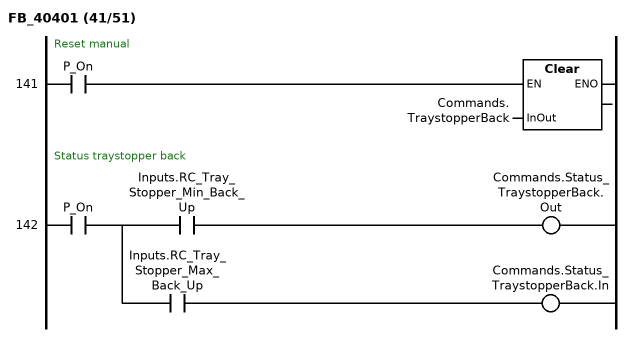
(* [picture p174: FB_40401, rungs 141-142] *)
(* Rung 141: Reset manual *)
IF P_On THEN Clear(InOut := Commands.TraystopperBack); END_IF;
(* Rung 142: Status traystopper back *)
Commands.Status_TraystopperBack.Out := P_On AND Inputs.RC_Tray_Stopper_Min_Back_Up;
Commands.Status_TraystopperBack.In := P_On AND Inputs.RC_Tray_Stopper_Max_Back_Up;

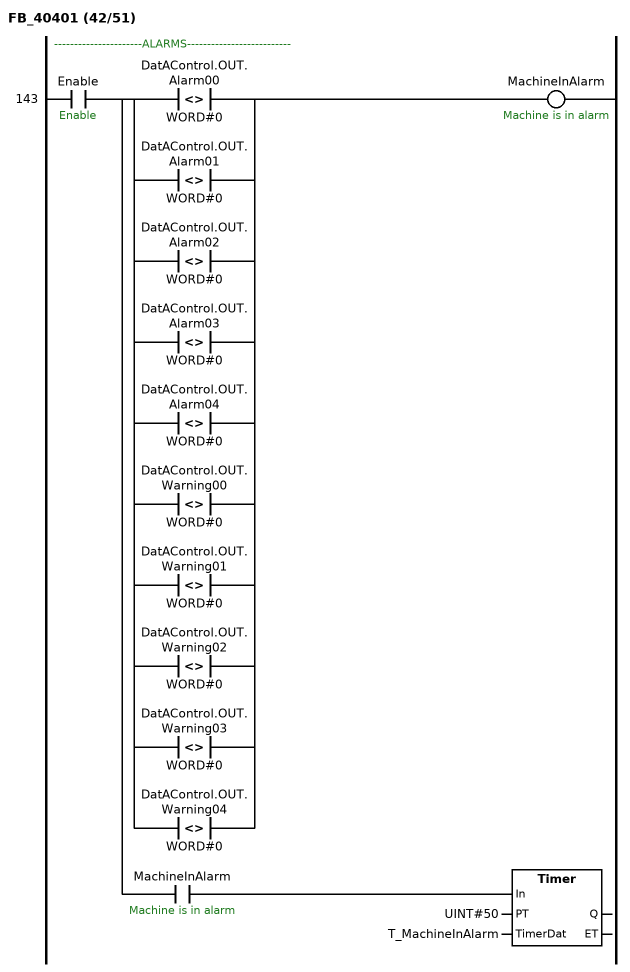
(* Rung 143: ----------------------ALARMS-------------------------- *)
MachineInAlarm := Enable AND ((DatAControl.OUT.Alarm00 <> WORD#0) OR (DatAControl.OUT.Alarm01 <> WORD#0) OR (DatAControl.OUT.Alarm02 <> WORD#0) OR (DatAControl.OUT.Alarm03 <> WORD#0) OR (DatAControl.OUT.Alarm04 <> WORD#0) OR (DatAControl.OUT.Warning00 <> WORD#0) OR (DatAControl.OUT.Warning01 <> WORD#0) OR (DatAControl.OUT.Warning02 <> WORD#0) OR (DatAControl.OUT.Warning03 <> WORD#0) OR (DatAControl.OUT.Warning04 <> WORD#0));
_t68 := Timer(In := Enable AND MachineInAlarm, PT := UINT#50, TimerDat := T_MachineInAlarm);

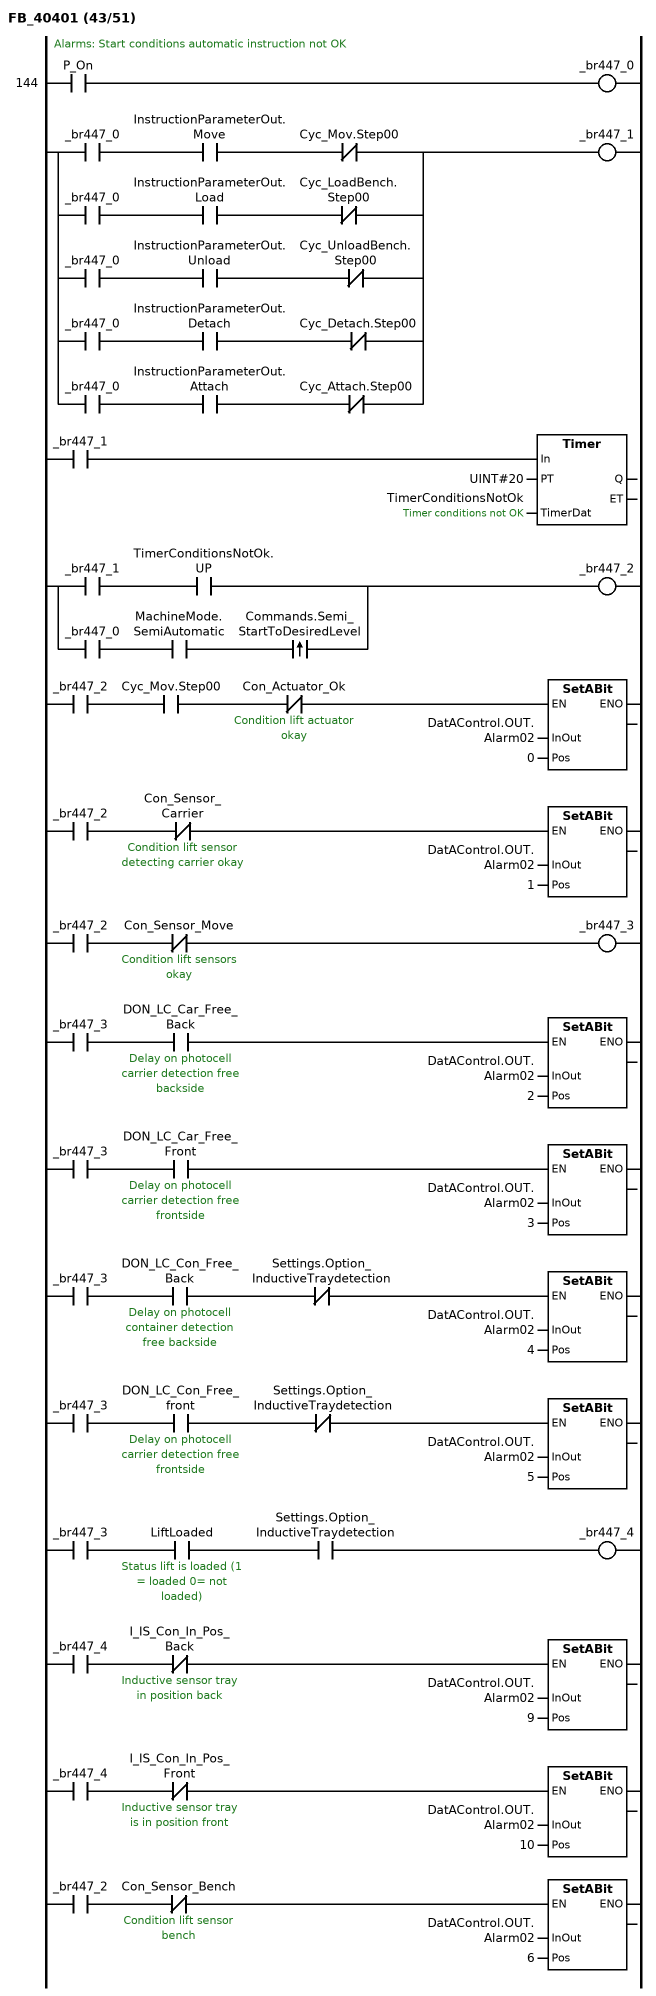
(* Rung 144: Alarms: Start conditions automatic instruction not OK *)
_br447_0 := P_On;
_br447_1 := (_br447_0 AND InstructionParameterOut.Move AND NOT Cyc_Mov.Step00) OR (_br447_0 AND InstructionParameterOut.Load AND NOT Cyc_LoadBench.Step00) OR (_br447_0 AND InstructionParameterOut.Unload AND NOT Cyc_UnloadBench.Step00) OR (_br447_0 AND InstructionParameterOut.Detach AND NOT Cyc_Detach.Step00) OR (_br447_0 AND InstructionParameterOut.Attach AND NOT Cyc_Attach.Step00);
_t69 := Timer(In := _br447_1, PT := UINT#20, TimerDat := TimerConditionsNotOk);
_e70(CLK := Commands.Semi_StartToDesiredLevel);
_br447_2 := (_br447_1 AND TimerConditionsNotOk.UP) OR (_br447_0 AND MachineMode.SemiAutomatic AND _e70.Q);
IF _br447_2 AND Cyc_Mov.Step00 AND NOT Con_Actuator_Ok THEN
    SetABit(InOut := DatAControl.OUT.Alarm02, Pos := 0);
END_IF;
IF _br447_2 AND NOT Con_Sensor_Carrier THEN SetABit(InOut := DatAControl.OUT.Alarm02, Pos := 1); END_IF;
_br447_3 := _br447_2 AND NOT Con_Sensor_Move;
IF _br447_3 AND DON_LC_Car_Free_Back THEN SetABit(InOut := DatAControl.OUT.Alarm02, Pos := 2); END_IF;
IF _br447_3 AND DON_LC_Car_Free_Front THEN SetABit(InOut := DatAControl.OUT.Alarm02, Pos := 3); END_IF;
IF _br447_3 AND DON_LC_Con_Free_Back AND NOT Settings.Option_InductiveTraydetection THEN
    SetABit(InOut := DatAControl.OUT.Alarm02, Pos := 4);
END_IF;
IF _br447_3 AND DON_LC_Con_Free_front AND NOT Settings.Option_InductiveTraydetection THEN
    SetABit(InOut := DatAControl.OUT.Alarm02, Pos := 5);
END_IF;
_br447_4 := _br447_3 AND LiftLoaded AND Settings.Option_InductiveTraydetection;
IF _br447_4 AND NOT I_IS_Con_In_Pos_Back THEN SetABit(InOut := DatAControl.OUT.Alarm02, Pos := 9); END_IF;
IF _br447_4 AND NOT I_IS_Con_In_Pos_Front THEN
    SetABit(InOut := DatAControl.OUT.Alarm02, Pos := 10);
END_IF;
IF _br447_2 AND NOT Con_Sensor_Bench THEN SetABit(InOut := DatAControl.OUT.Alarm02, Pos := 6); END_IF;

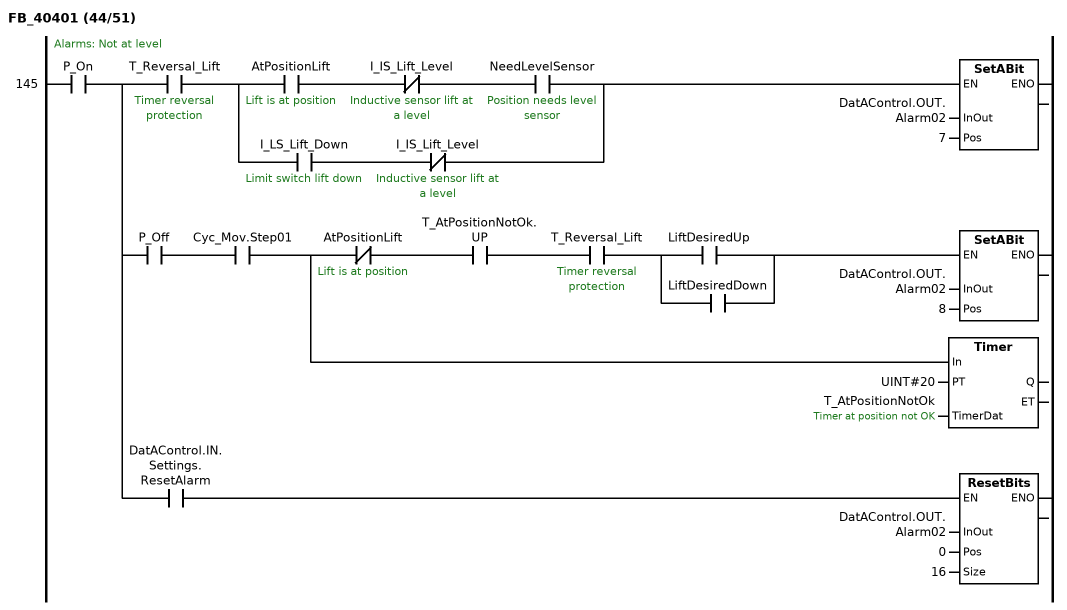
(* Rung 145: Alarms: Not at level *)
IF P_On AND T_Reversal_Lift AND ((AtPositionLift AND NOT I_IS_Lift_Level AND NeedLevelSensor) OR (I_LS_Lift_Down AND NOT I_IS_Lift_Level)) THEN
    SetABit(InOut := DatAControl.OUT.Alarm02, Pos := 7);
END_IF;
IF P_On AND P_Off AND Cyc_Mov.Step01 AND NOT AtPositionLift AND T_AtPositionNotOk.UP AND T_Reversal_Lift AND (LiftDesiredUp OR LiftDesiredDown) THEN
    SetABit(InOut := DatAControl.OUT.Alarm02, Pos := 8);
END_IF;
_t71 := Timer(In := P_On AND P_Off AND Cyc_Mov.Step01, PT := UINT#20, TimerDat := T_AtPositionNotOk);
IF P_On AND DatAControl.IN.Settings.ResetAlarm THEN
    ResetBits(InOut := DatAControl.OUT.Alarm02, Pos := 0, Size := 16);
END_IF;

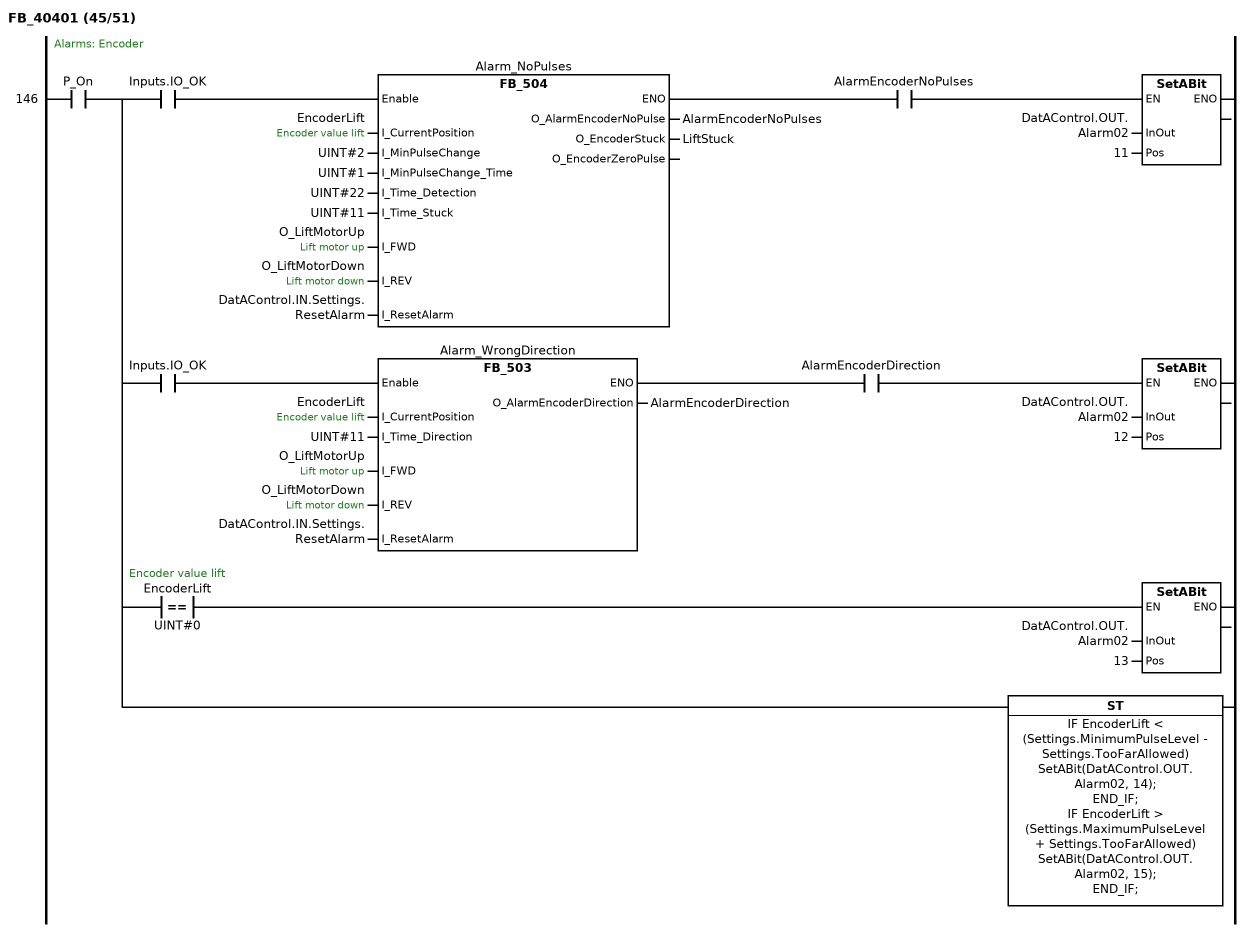
(* Rung 146: Alarms: Encoder *)
Alarm_NoPulses(Enable := P_On AND Inputs.IO_OK, I_CurrentPosition := EncoderLift, I_MinPulseChange := UINT#2, I_MinPulseChange_Time := UINT#1, I_Time_Detection := UINT#22, I_Time_Stuck := UINT#11, I_FWD := O_LiftMotorUp, I_REV := O_LiftMotorDown, I_ResetAlarm := DatAControl.IN.Settings.ResetAlarm, O_AlarmEncoderNoPulse => AlarmEncoderNoPulses, O_EncoderStuck => LiftStuck);
IF Alarm_NoPulses.ENO AND AlarmEncoderNoPulses THEN
    SetABit(InOut := DatAControl.OUT.Alarm02, Pos := 11);
END_IF;
Alarm_WrongDirection(Enable := P_On AND Inputs.IO_OK, I_CurrentPosition := EncoderLift, I_Time_Direction := UINT#11, I_FWD := O_LiftMotorUp, I_REV := O_LiftMotorDown, I_ResetAlarm := DatAControl.IN.Settings.ResetAlarm, O_AlarmEncoderDirection => AlarmEncoderDirection);
IF Alarm_WrongDirection.ENO AND AlarmEncoderDirection THEN
    SetABit(InOut := DatAControl.OUT.Alarm02, Pos := 12);
END_IF;
IF P_On AND (EncoderLift = UINT#0) THEN SetABit(InOut := DatAControl.OUT.Alarm02, Pos := 13); END_IF;
IF P_On THEN
    IF EncoderLift < (Settings.MinimumPulseLevel - Settings.TooFarAllowed) THEN
    	SetABit(DatAControl.OUT.Alarm02, 14);
    END_IF;
    
    IF EncoderLift > (Settings.MaximumPulseLevel + Settings.TooFarAllowed) THEN
    	SetABit(DatAControl.OUT.Alarm02, 15);
    END_IF;
END_IF;

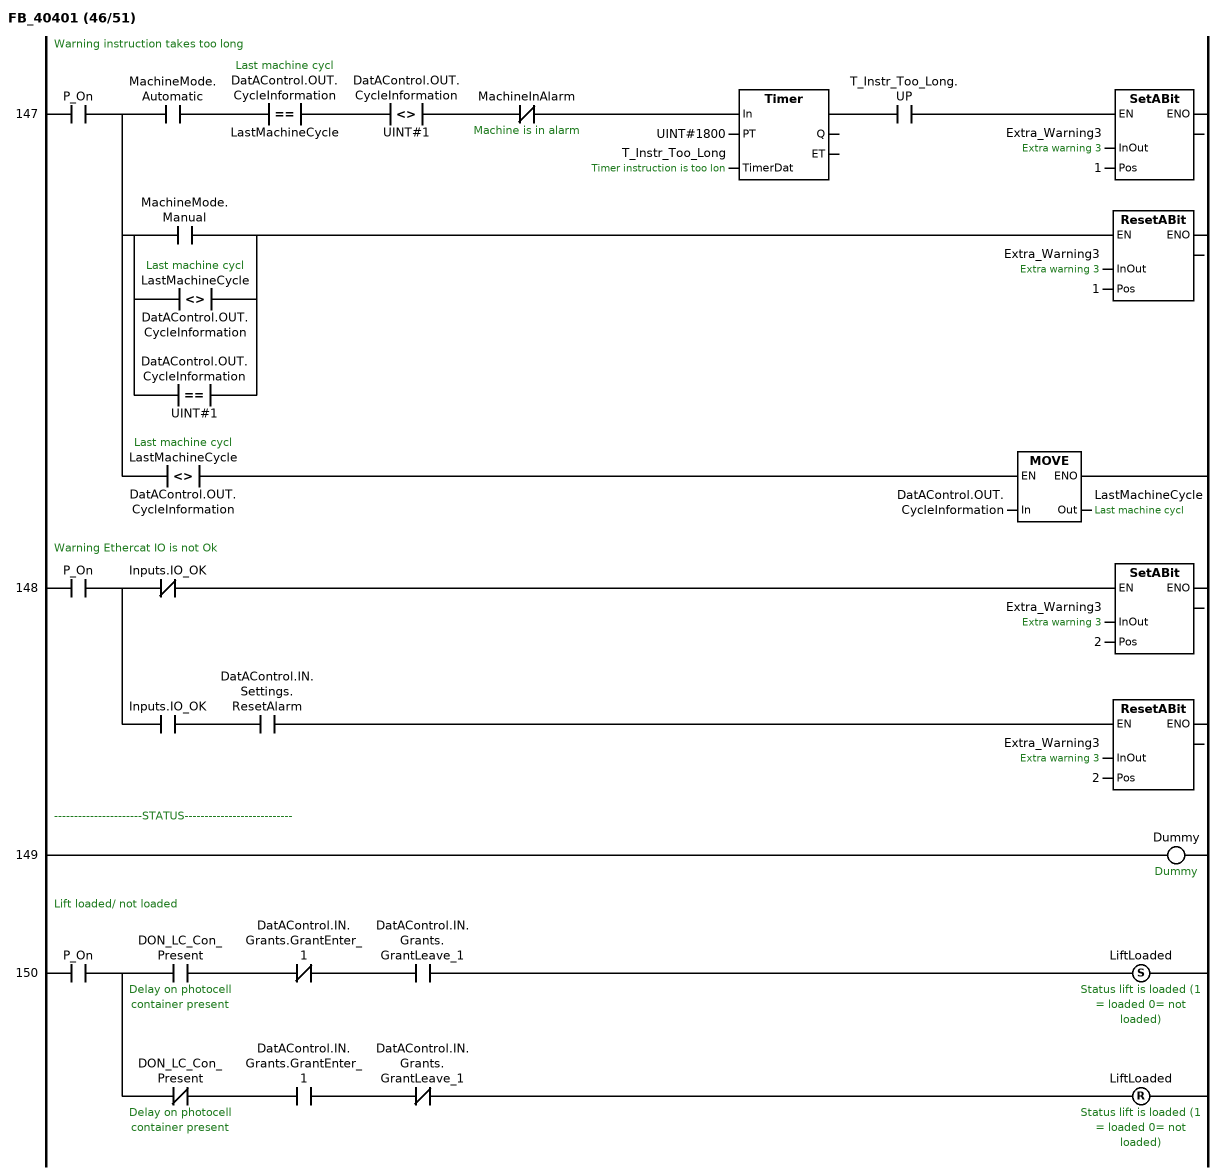
(* Rung 147: Warning instruction takes too long *)
_p73 := P_On AND MachineMode.Automatic AND (DatAControl.OUT.CycleInformation = LastMachineCycle) AND (DatAControl.OUT.CycleInformation <> UINT#1) AND NOT MachineInAlarm;
_t72 := Timer(In := _p73, PT := UINT#1800, TimerDat := T_Instr_Too_Long);
IF _t72 AND T_Instr_Too_Long.UP THEN SetABit(InOut := Extra_Warning3, Pos := 1); END_IF;
IF P_On AND (MachineMode.Manual OR (LastMachineCycle <> DatAControl.OUT.CycleInformation) OR (DatAControl.OUT.CycleInformation = UINT#1)) THEN
    ResetABit(InOut := Extra_Warning3, Pos := 1);
END_IF;
IF P_On AND (LastMachineCycle <> DatAControl.OUT.CycleInformation) THEN
    LastMachineCycle := DatAControl.OUT.CycleInformation;
END_IF;
(* Rung 148: Warning Ethercat IO is not Ok *)
IF P_On AND NOT Inputs.IO_OK THEN SetABit(InOut := Extra_Warning3, Pos := 2); END_IF;
IF P_On AND Inputs.IO_OK AND DatAControl.IN.Settings.ResetAlarm THEN
    ResetABit(InOut := Extra_Warning3, Pos := 2);
END_IF;
(* Rung 149: ----------------------STATUS--------------------------- *)
Dummy := TRUE;
(* Rung 150: Lift loaded/ not loaded *)
IF P_On AND DON_LC_Con_Present AND NOT DatAControl.IN.Grants.GrantEnter_1 AND DatAControl.IN.Grants.GrantLeave_1 THEN
    LiftLoaded := TRUE;
END_IF;
IF P_On AND NOT DON_LC_Con_Present AND DatAControl.IN.Grants.GrantEnter_1 AND NOT DatAControl.IN.Grants.GrantLeave_1 THEN
    LiftLoaded := FALSE;
END_IF;

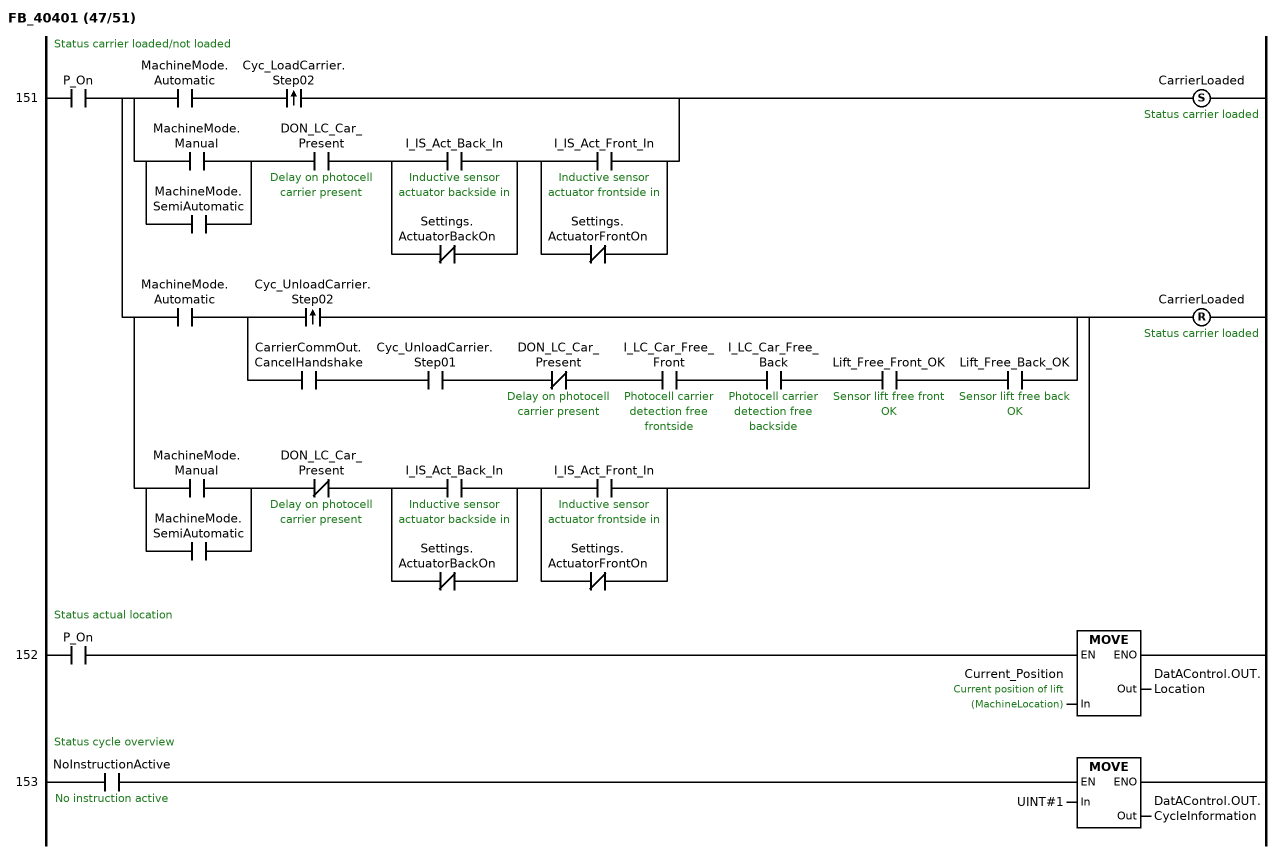
(* Rung 151: Status carrier loaded/not loaded *)
_e74(CLK := Cyc_LoadCarrier.Step02);
IF P_On AND ((MachineMode.Automatic AND _e74.Q) OR ((MachineMode.Manual OR MachineMode.SemiAutomatic) AND DON_LC_Car_Present AND (I_IS_Act_Back_In OR NOT Settings.ActuatorBackOn) AND (I_IS_Act_Front_In OR NOT Settings.ActuatorFrontOn))) THEN
    CarrierLoaded := TRUE;
END_IF;
_e75(CLK := Cyc_UnloadCarrier.Step02);
IF P_On AND ((MachineMode.Automatic AND (_e75.Q OR (CarrierCommOut.CancelHandshake AND Cyc_UnloadCarrier.Step01 AND NOT DON_LC_Car_Present AND I_LC_Car_Free_Front AND I_LC_Car_Free_Back AND Lift_Free_Front_OK AND Lift_Free_Back_OK))) OR ((MachineMode.Manual OR MachineMode.SemiAutomatic) AND NOT DON_LC_Car_Present AND (I_IS_Act_Back_In OR NOT Settings.ActuatorBackOn) AND (I_IS_Act_Front_In OR NOT Settings.ActuatorFrontOn))) THEN
    CarrierLoaded := FALSE;
END_IF;
(* Rung 152: Status actual location *)
IF P_On THEN DatAControl.OUT.Location := Current_Position; END_IF;
(* Rung 153: Status cycle overview *)
IF NoInstructionActive THEN DatAControl.OUT.CycleInformation := UINT#1; END_IF;

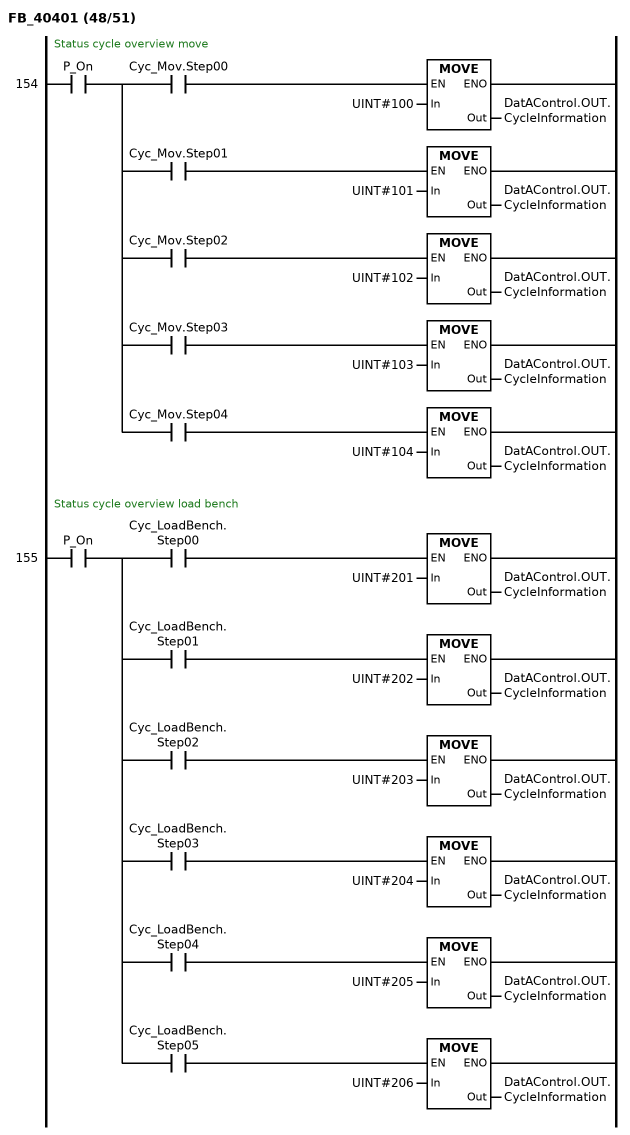
(* Rung 154: Status cycle overview move *)
IF P_On AND Cyc_Mov.Step00 THEN DatAControl.OUT.CycleInformation := UINT#100; END_IF;
IF P_On AND Cyc_Mov.Step01 THEN DatAControl.OUT.CycleInformation := UINT#101; END_IF;
IF P_On AND Cyc_Mov.Step02 THEN DatAControl.OUT.CycleInformation := UINT#102; END_IF;
IF P_On AND Cyc_Mov.Step03 THEN DatAControl.OUT.CycleInformation := UINT#103; END_IF;
IF P_On AND Cyc_Mov.Step04 THEN DatAControl.OUT.CycleInformation := UINT#104; END_IF;
(* Rung 155: Status cycle overview load bench *)
IF P_On AND Cyc_LoadBench.Step00 THEN DatAControl.OUT.CycleInformation := UINT#201; END_IF;
IF P_On AND Cyc_LoadBench.Step01 THEN DatAControl.OUT.CycleInformation := UINT#202; END_IF;
IF P_On AND Cyc_LoadBench.Step02 THEN DatAControl.OUT.CycleInformation := UINT#203; END_IF;
IF P_On AND Cyc_LoadBench.Step03 THEN DatAControl.OUT.CycleInformation := UINT#204; END_IF;
IF P_On AND Cyc_LoadBench.Step04 THEN DatAControl.OUT.CycleInformation := UINT#205; END_IF;
IF P_On AND Cyc_LoadBench.Step05 THEN DatAControl.OUT.CycleInformation := UINT#206; END_IF;

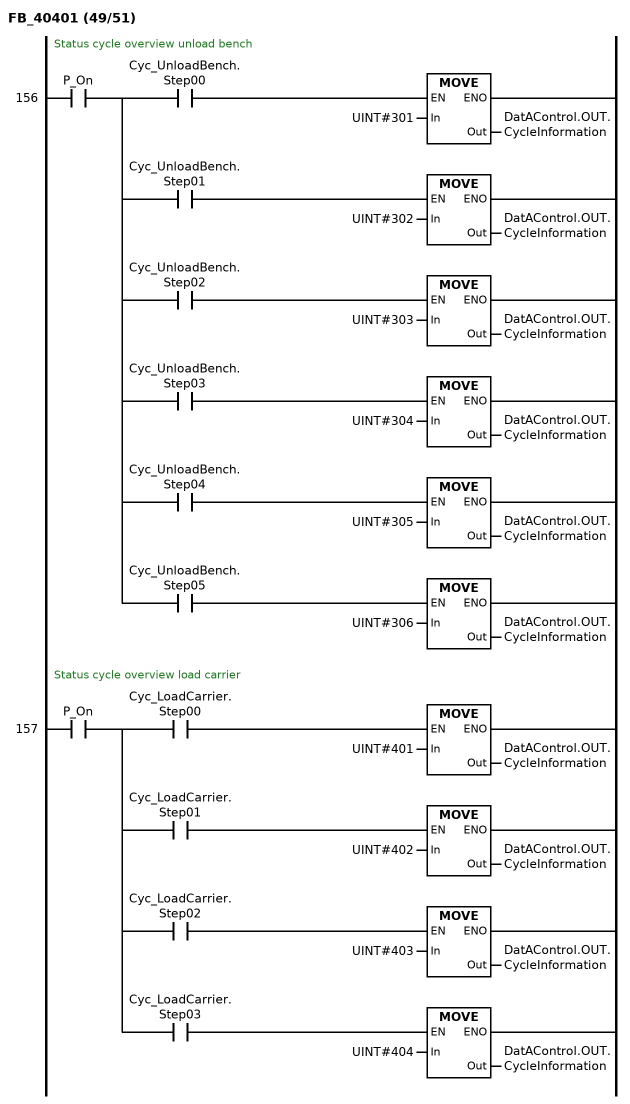
(* Rung 156: Status cycle overview unload bench *)
IF P_On AND Cyc_UnloadBench.Step00 THEN DatAControl.OUT.CycleInformation := UINT#301; END_IF;
IF P_On AND Cyc_UnloadBench.Step01 THEN DatAControl.OUT.CycleInformation := UINT#302; END_IF;
IF P_On AND Cyc_UnloadBench.Step02 THEN DatAControl.OUT.CycleInformation := UINT#303; END_IF;
IF P_On AND Cyc_UnloadBench.Step03 THEN DatAControl.OUT.CycleInformation := UINT#304; END_IF;
IF P_On AND Cyc_UnloadBench.Step04 THEN DatAControl.OUT.CycleInformation := UINT#305; END_IF;
IF P_On AND Cyc_UnloadBench.Step05 THEN DatAControl.OUT.CycleInformation := UINT#306; END_IF;
(* Rung 157: Status cycle overview load carrier *)
IF P_On AND Cyc_LoadCarrier.Step00 THEN DatAControl.OUT.CycleInformation := UINT#401; END_IF;
IF P_On AND Cyc_LoadCarrier.Step01 THEN DatAControl.OUT.CycleInformation := UINT#402; END_IF;
IF P_On AND Cyc_LoadCarrier.Step02 THEN DatAControl.OUT.CycleInformation := UINT#403; END_IF;
IF P_On AND Cyc_LoadCarrier.Step03 THEN DatAControl.OUT.CycleInformation := UINT#404; END_IF;

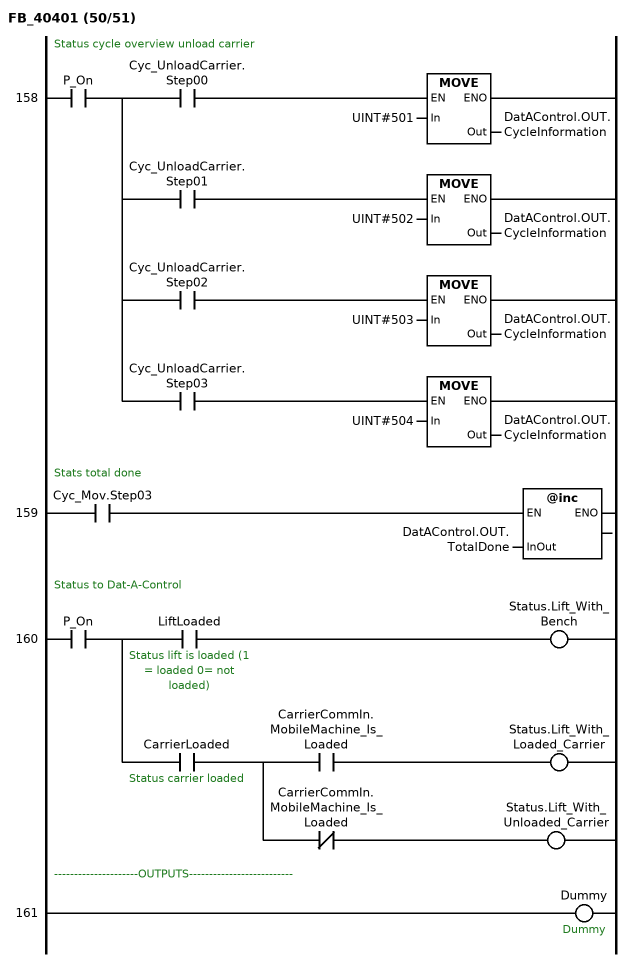
(* Rung 158: Status cycle overview unload carrier *)
IF P_On AND Cyc_UnloadCarrier.Step00 THEN DatAControl.OUT.CycleInformation := UINT#501; END_IF;
IF P_On AND Cyc_UnloadCarrier.Step01 THEN DatAControl.OUT.CycleInformation := UINT#502; END_IF;
IF P_On AND Cyc_UnloadCarrier.Step02 THEN DatAControl.OUT.CycleInformation := UINT#503; END_IF;
IF P_On AND Cyc_UnloadCarrier.Step03 THEN DatAControl.OUT.CycleInformation := UINT#504; END_IF;
(* Rung 159: Stats total done *)
_e76(CLK := Cyc_Mov.Step03);
IF _e76.Q THEN inc(InOut := DatAControl.OUT.TotalDone); END_IF;
(* Rung 160: Status to Dat-A-Control *)
Status.Lift_With_Bench := P_On AND LiftLoaded;
Status.Lift_With_Loaded_Carrier := P_On AND CarrierLoaded AND CarrierCommIn.MobileMachine_Is_Loaded;
Status.Lift_With_Unloaded_Carrier := P_On AND CarrierLoaded AND NOT CarrierCommIn.MobileMachine_Is_Loaded;
(* Rung 161: ---------------------OUTPUTS-------------------------- *)
Dummy := TRUE;

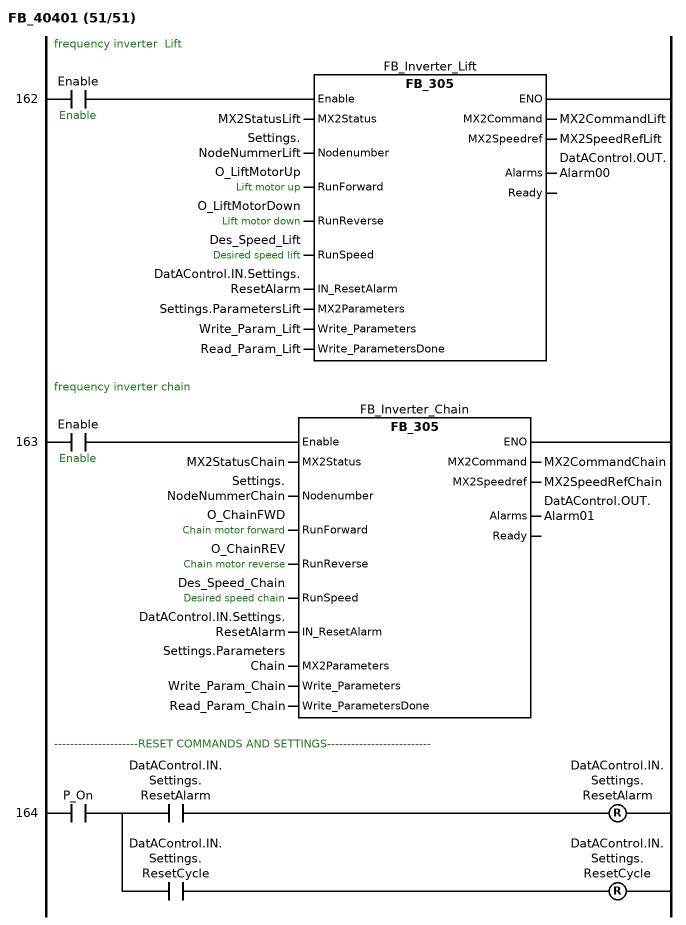
(* Rung 162: frequency inverter  Lift *)
FB_Inverter_Lift(Enable := Enable, MX2Status := MX2StatusLift, Nodenumber := Settings.NodeNummerLift, RunForward := O_LiftMotorUp, RunReverse := O_LiftMotorDown, RunSpeed := Des_Speed_Lift, IN_ResetAlarm := DatAControl.IN.Settings.ResetAlarm, MX2Parameters := Settings.ParametersLift, Write_Parameters := Write_Param_Lift, Write_ParametersDone := Read_Param_Lift, MX2Command => MX2CommandLift, MX2Speedref => MX2SpeedRefLift, Alarms => DatAControl.OUT.Alarm00);
(* Rung 163: frequency inverter chain *)
FB_Inverter_Chain(Enable := Enable, MX2Status := MX2StatusChain, Nodenumber := Settings.NodeNummerChain, RunForward := O_ChainFWD, RunReverse := O_ChainREV, RunSpeed := Des_Speed_Chain, IN_ResetAlarm := DatAControl.IN.Settings.ResetAlarm, MX2Parameters := Settings.ParametersChain, Write_Parameters := Write_Param_Chain, Write_ParametersDone := Read_Param_Chain, MX2Command => MX2CommandChain, MX2Speedref => MX2SpeedRefChain, Alarms => DatAControl.OUT.Alarm01);
(* Rung 164: ---------------------RESET COMMANDS AND SETTINGS-------------------------- *)
IF P_On AND DatAControl.IN.Settings.ResetAlarm THEN DatAControl.IN.Settings.ResetAlarm := FALSE; END_IF;
IF P_On AND DatAControl.IN.Settings.ResetCycle THEN DatAControl.IN.Settings.ResetCycle := FALSE; END_IF;
END_FUNCTION_BLOCK

FUNCTION_BLOCK FB_40303
VAR RETAIN
    Cyc_Turning : ST_FB_40303_Cycle_Turning;  (* Step01 Close clamps; Step02 Lift from middle to up; Step00 Request for cleaning, lift from down to middle; Step03 Lift is up, ready to clean; Step04 Lift from up to middle; Step05 Open clamps; Step06 Lift from middle to down; Step07 Lift is down, clean cycle is ready *)
    Cyc_Cleaning : ST_FB_40303_Cycle_Cleaning;  (* Step02 Move sprayboom to left side for gutter cleaning *)
END_VAR
VAR
    Dummy : BOOL;  (* Dummy *)
    NoAlarms : BOOL;  (* There are currently no alarms *)
    T_PowerOK : _sTimer;  (* Timer power OK *)
    Release : BOOL;  (* Release according to emergency stop and alarms *)
    MachineMode : ST_MachineMode;  (* Machine mode *)
    FB_Inverter_TurningFrame : FB_305;
    FB_Inverter_SprayBoom : FB_305;
    FB_Inverter_DirtBelt : FB_305;
    TurningFrame_Forward : BOOL;  (* Turningframe run forward *)
    TurningFrame_Backward : BOOL;  (* Turningframe run backward *)
    SprayBoom_Forward : BOOL;  (* Sprayboom forward to the left *)
    SprayBoom_Backward : BOOL;  (* Sprayboom backward to the right *)
    DirtBelt_Forward : BOOL;  (* Dirtbelt run forward *)
    DirtBelt_Backward : BOOL;  (* Dirtbelt run backward *)
    TurningFrame_Down_Don : BOOL;  (* Turningframe down delayed on *)
    TurningFrame_Middle_Don : BOOL;  (* Turningframe middle delayed on *)
    TurningFrame_Up_Don : BOOL;  (* Turningframe up delayed on *)
    Clamps_Loose_Don : BOOL;  (* Clamps loose delayed on *)
    Clamps_Fixed_Don : BOOL;  (* Clamps fixed delayed on *)
    FB_Clamps : FB_1017;
    Condition_Clamps : BOOL;  (* Global condition to move the clamps *)
    ManualControl_Clamps : ST_ManualControl_Actuator;  (* Manual control clamps *)
    Reference_Clamps : UINT;  (* Reference (1=fixed, 2=loose) *)
    AmountMovements_Clamps : UDINT;  (* Amount of movements clamps *)
    Alarms_Clamps : BYTE;  (* Alarm clamps *)
    Warnings_Clamps : BYTE;  (* Warnings clamps *)
    FB_Dirtbelt : FB_1011;
    LetDirtbeltRun : BOOL;  (* Let dirtbelt run *)
END_VAR
VAR RETAIN
    AmountMovements_DirtBelt : UDINT;  (* Amount of movements dirtbelt *)
END_VAR
VAR
    Alarms_Dirtbelt : BYTE;  (* Alarms dirtbelt *)
    FB_SprayBoom : FB_1014;
    Condition_SprayBoom : BOOL;  (* Global condition to move the sprayboom *)
    T_Dirtbelt_RunLonger : _sTimer;  (* Timer let dirtbelt run longer after spraying *)
    FB_TurningFrame : FB_1018;
    Condition_TurningFrame : BOOL;  (* Global condition to move the turningframe *)
    ManualControl_TurningFrame : ST_ManualControl_Actuator;  (* Manual control turningframe *)
    Reference_TurningFrame : UINT;  (* Reference (1=down, 2=middle, 3=up) *)
    TurningFrameSpeed : UINT;  (* Speed for turningframe *)
    Alarms_TurningFrame : BYTE;  (* Alarms turningframe *)
    AmountMovements_TurningFrame : UDINT;  (* Amount of movements turningframe *)
    SprayBoom_Right_Don : BOOL;  (* Sprayboom at the right delayed on *)
    SprayBoom_Left_Don : BOOL;  (* Sprayboom at the left delayed on *)
    AmountMovements_SprayBoom : UDINT;  (* Amount of movements sprayboom *)
    Alarms_SprayBoom : BYTE;  (* Alarms sprayboom *)
    Warnings_SprayBoom : BYTE;  (* Warnings sprayboom *)
    ManualControl_SprayBoom : ST_ManualControl_Actuator;
    Reference_SprayBoom : UINT;  (* Reference (1=right, 2=left) *)
    Alarms_Inverter_TurningFrame : BYTE;  (* Alarms inverter turningframe *)
    Alarms_Inverter_SprayBoom : BYTE;  (* Alarms inverter sprayboom *)
    Alarms_Inverter_Dirtbelt : BYTE;  (* Alarms inverter dirtbelt *)
    T_PressureSprayboomMain_Off : _sTimer;  (* Timer pressure is low enough sprayboom *)
    T_PressureSprayboomMain_On : _sTimer;  (* Timer pressure is high enough sprayboom *)
    Desired_Amount_Sprayboom : UDINT;
    T_CleanGutterLeft : _sTimer;
    T_CleanGutterRight : _sTimer;
END_VAR
VAR_INPUT
    Enable : BOOL;  (* Enable *)
    Status_dirtbelt : ST_MX2\Status;
    Status_SprayBoom : ST_MX2\Status;
    Status_TurningFrame : ST_MX2\Status;
    Inputs : ST_FB_40303_Inputs;  (* Inputs *)
    Settings : ST_FB_40303_Settings;  (* Settings *)
    StartWashCycle : BOOL;  (* Start wash cycle *)
    WashCycleReadyOK : BOOL;  (* Wash cycle ready OK *)
END_VAR
VAR_OUTPUT
    Outputs : ST_FB_40303_Outputs;  (* Outputs; S_FillCleanWater Outputs fill clean water *)
    ReleaseTransport : BOOL;  (* Output to external system: Release for container transport *)
    WashCycleReady : BOOL;  (* Output to external system: Wash cycle ready *)
END_VAR
VAR_IN_OUT
    DatAControl : ST_DatAControl_Standard;  (* Dat-A-Control *)
    Commands : ST_FB_40303_Commands;  (* Commands *)
    StatusContainer : BOOL;  (* Status container in cleaner (0 = clean, 1 = dirty) *)
    InverterTurningFrame_WriteParameters : BOOL;  (* Write parameters *)
    InverterTurningFrame_WriteParametersDone : BOOL;  (* Write parameters done *)
    InverterSprayboom_WriteParameters : BOOL;  (* Write parameters *)
    InverterSprayboom_WriteParametersDone : BOOL;  (* Write parameters done *)
    InverterDirtBelt_WriteParameters : BOOL;  (* Write parameters *)
    InverterDirtBelt_WriteParametersDone : BOOL;  (* Write parameters done *)
END_VAR
VAR
    _t1 : BOOL;
    _t2 : BOOL;
    _p3 : BOOL;
    _e4 : R_TRIG;
    _e5 : R_TRIG;
    _e6 : R_TRIG;
    _p7 : BOOL;
    _t8 : BOOL;
    _e9 : R_TRIG;
    _p10 : BOOL;
    _t11 : BOOL;
    _e12 : R_TRIG;
    _p13 : BOOL;
    _e14 : R_TRIG;
    _e15 : R_TRIG;
    _t16 : BOOL;
    _t17 : BOOL;
    _t18 : BOOL;
END_VAR
(* ladder, written here as Structured Text *)

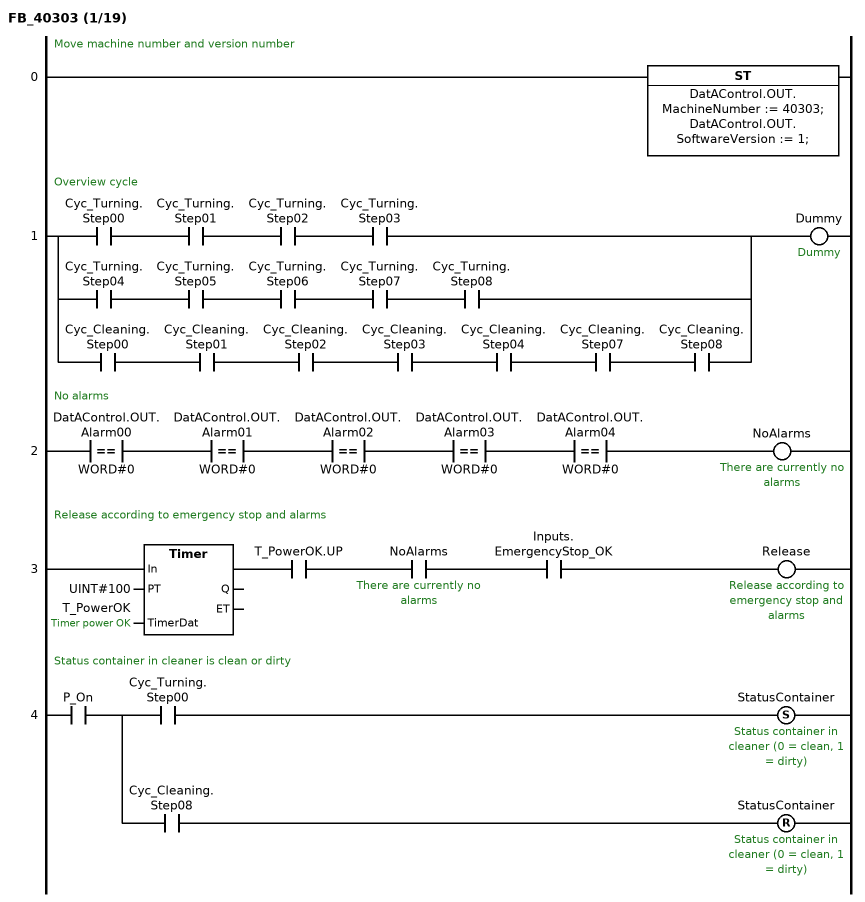
(* Rung 0: Move machine number and version number *)
DatAControl.OUT.MachineNumber := 40303;
DatAControl.OUT.SoftwareVersion := 1;
(* Rung 1: Overview cycle *)
Dummy := (Cyc_Turning.Step00 AND Cyc_Turning.Step01 AND Cyc_Turning.Step02 AND Cyc_Turning.Step03) OR (Cyc_Turning.Step04 AND Cyc_Turning.Step05 AND Cyc_Turning.Step06 AND Cyc_Turning.Step07 AND Cyc_Turning.Step08) OR (Cyc_Cleaning.Step00 AND Cyc_Cleaning.Step01 AND Cyc_Cleaning.Step02 AND Cyc_Cleaning.Step03 AND Cyc_Cleaning.Step04 AND Cyc_Cleaning.Step07 AND Cyc_Cleaning.Step08);
(* Rung 2: No alarms *)
NoAlarms := (DatAControl.OUT.Alarm00 = WORD#0) AND (DatAControl.OUT.Alarm01 = WORD#0) AND (DatAControl.OUT.Alarm02 = WORD#0) AND (DatAControl.OUT.Alarm03 = WORD#0) AND (DatAControl.OUT.Alarm04 = WORD#0);
(* Rung 3: Release according to emergency stop and alarms *)
_t1 := Timer(In := TRUE, PT := UINT#100, TimerDat := T_PowerOK);
Release := _t1 AND T_PowerOK.UP AND NoAlarms AND Inputs.EmergencyStop_OK;
(* Rung 4: Status container in cleaner is clean or dirty *)
IF P_On AND Cyc_Turning.Step00 THEN StatusContainer := TRUE; END_IF;
IF P_On AND Cyc_Cleaning.Step08 THEN StatusContainer := FALSE; END_IF;

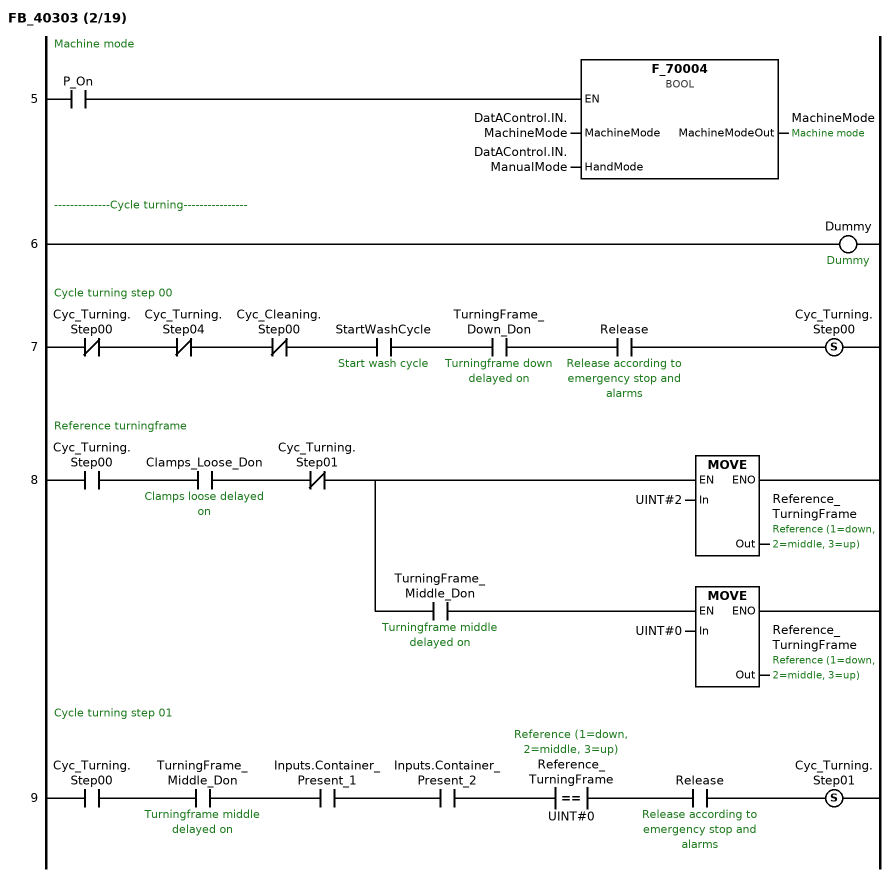
(* Rung 5: Machine mode *)
_t2 := FALSE;
IF P_On THEN _t2 := F_70004(MachineMode := DatAControl.IN.MachineMode, HandMode := DatAControl.IN.ManualMode, MachineModeOut => MachineMode); END_IF;
(* Rung 6: --------------Cycle turning---------------- *)
Dummy := TRUE;
(* Rung 7: Cycle turning step 00 *)
IF NOT Cyc_Turning.Step00 AND NOT Cyc_Turning.Step04 AND NOT Cyc_Cleaning.Step00 AND StartWashCycle AND TurningFrame_Down_Don AND Release THEN
    Cyc_Turning.Step00 := TRUE;
END_IF;
(* Rung 8: Reference turningframe *)
_p3 := Cyc_Turning.Step00 AND Clamps_Loose_Don AND NOT Cyc_Turning.Step01;
IF _p3 THEN Reference_TurningFrame := UINT#2; END_IF;
IF _p3 AND TurningFrame_Middle_Don THEN Reference_TurningFrame := UINT#0; END_IF;
(* Rung 9: Cycle turning step 01 *)
IF Cyc_Turning.Step00 AND TurningFrame_Middle_Don AND Inputs.Container_Present_1 AND Inputs.Container_Present_2 AND (Reference_TurningFrame = UINT#0) AND Release THEN
    Cyc_Turning.Step01 := TRUE;
END_IF;

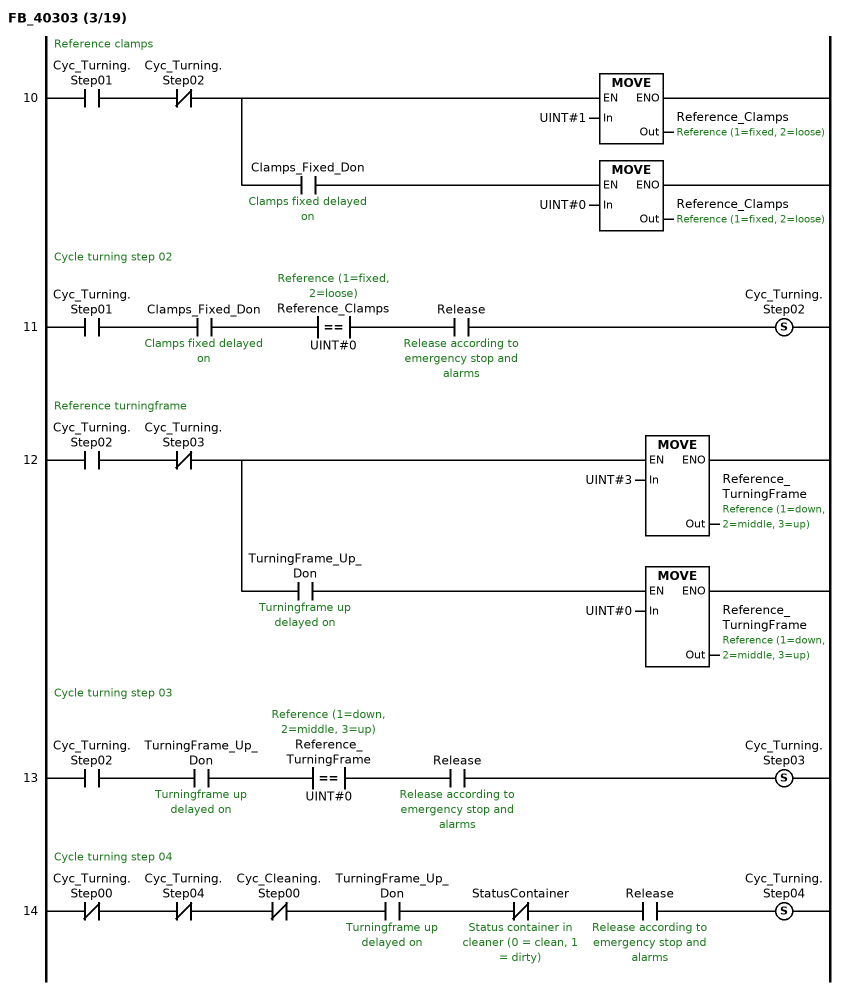
(* Rung 10: Reference clamps *)
IF Cyc_Turning.Step01 AND NOT Cyc_Turning.Step02 THEN Reference_Clamps := UINT#1; END_IF;
IF Cyc_Turning.Step01 AND NOT Cyc_Turning.Step02 AND Clamps_Fixed_Don THEN
    Reference_Clamps := UINT#0;
END_IF;
(* Rung 11: Cycle turning step 02 *)
IF Cyc_Turning.Step01 AND Clamps_Fixed_Don AND (Reference_Clamps = UINT#0) AND Release THEN
    Cyc_Turning.Step02 := TRUE;
END_IF;
(* Rung 12: Reference turningframe *)
IF Cyc_Turning.Step02 AND NOT Cyc_Turning.Step03 THEN Reference_TurningFrame := UINT#3; END_IF;
IF Cyc_Turning.Step02 AND NOT Cyc_Turning.Step03 AND TurningFrame_Up_Don THEN
    Reference_TurningFrame := UINT#0;
END_IF;
(* Rung 13: Cycle turning step 03 *)
IF Cyc_Turning.Step02 AND TurningFrame_Up_Don AND (Reference_TurningFrame = UINT#0) AND Release THEN
    Cyc_Turning.Step03 := TRUE;
END_IF;
(* Rung 14: Cycle turning step 04 *)
IF NOT Cyc_Turning.Step00 AND NOT Cyc_Turning.Step04 AND NOT Cyc_Cleaning.Step00 AND TurningFrame_Up_Don AND NOT StatusContainer AND Release THEN
    Cyc_Turning.Step04 := TRUE;
END_IF;

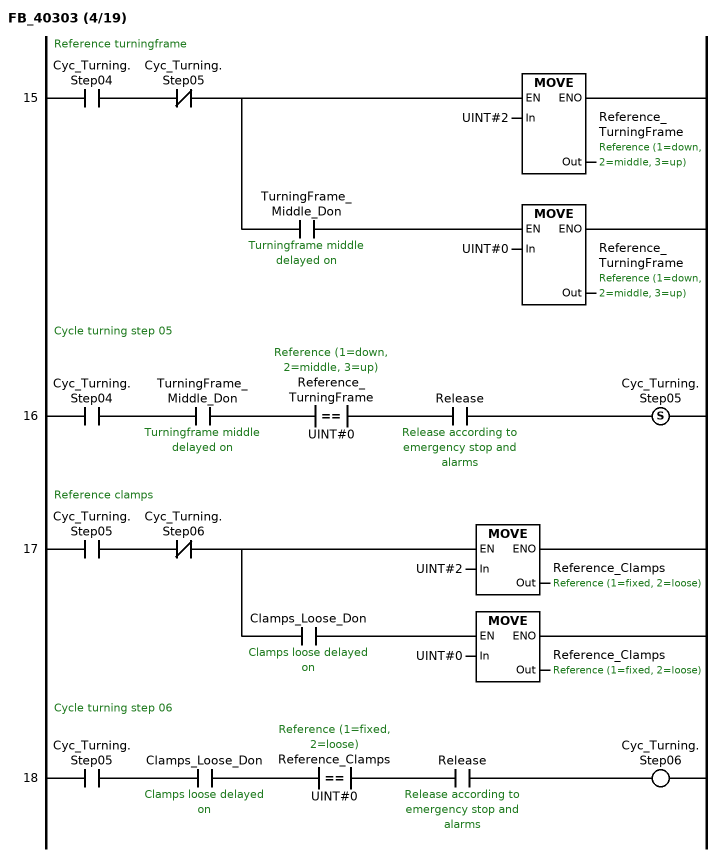
(* Rung 15: Reference turningframe *)
IF Cyc_Turning.Step04 AND NOT Cyc_Turning.Step05 THEN Reference_TurningFrame := UINT#2; END_IF;
IF Cyc_Turning.Step04 AND NOT Cyc_Turning.Step05 AND TurningFrame_Middle_Don THEN
    Reference_TurningFrame := UINT#0;
END_IF;
(* Rung 16: Cycle turning step 05 *)
IF Cyc_Turning.Step04 AND TurningFrame_Middle_Don AND (Reference_TurningFrame = UINT#0) AND Release THEN
    Cyc_Turning.Step05 := TRUE;
END_IF;
(* Rung 17: Reference clamps *)
IF Cyc_Turning.Step05 AND NOT Cyc_Turning.Step06 THEN Reference_Clamps := UINT#2; END_IF;
IF Cyc_Turning.Step05 AND NOT Cyc_Turning.Step06 AND Clamps_Loose_Don THEN
    Reference_Clamps := UINT#0;
END_IF;
(* Rung 18: Cycle turning step 06 *)
Cyc_Turning.Step06 := Cyc_Turning.Step05 AND Clamps_Loose_Don AND (Reference_Clamps = UINT#0) AND Release;

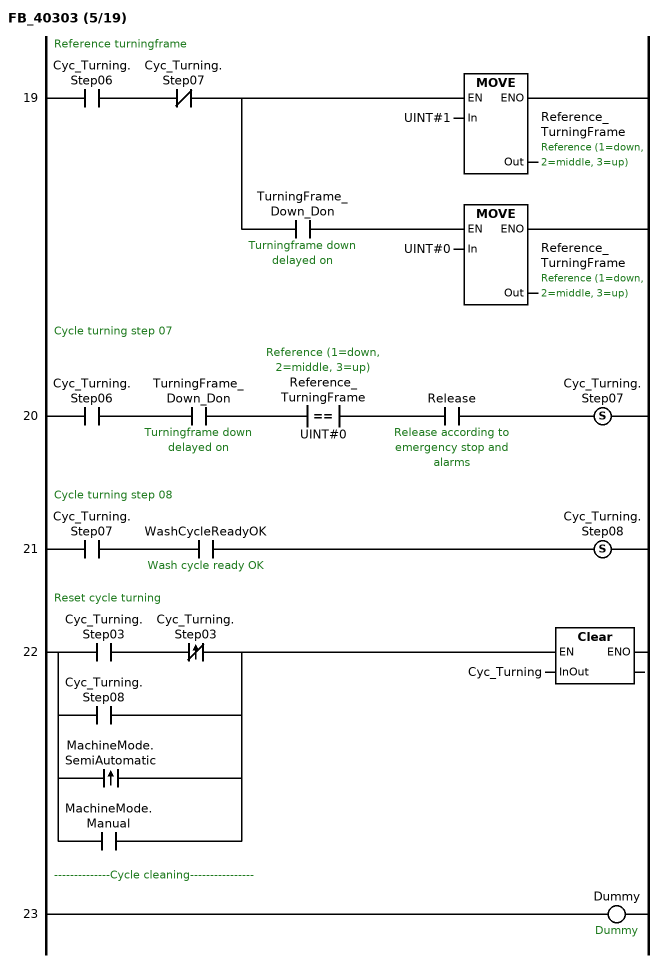
(* Rung 19: Reference turningframe *)
IF Cyc_Turning.Step06 AND NOT Cyc_Turning.Step07 THEN Reference_TurningFrame := UINT#1; END_IF;
IF Cyc_Turning.Step06 AND NOT Cyc_Turning.Step07 AND TurningFrame_Down_Don THEN
    Reference_TurningFrame := UINT#0;
END_IF;
(* Rung 20: Cycle turning step 07 *)
IF Cyc_Turning.Step06 AND TurningFrame_Down_Don AND (Reference_TurningFrame = UINT#0) AND Release THEN
    Cyc_Turning.Step07 := TRUE;
END_IF;
(* Rung 21: Cycle turning step 08 *)
IF Cyc_Turning.Step07 AND WashCycleReadyOK THEN Cyc_Turning.Step08 := TRUE; END_IF;
(* Rung 22: Reset cycle turning *)
_e4(CLK := Cyc_Turning.Step03);
_e5(CLK := MachineMode.SemiAutomatic);
IF (Cyc_Turning.Step03 AND NOT _e4.Q) OR Cyc_Turning.Step08 OR _e5.Q OR MachineMode.Manual THEN
    Clear(InOut := Cyc_Turning);
END_IF;
(* Rung 23: --------------Cycle cleaning---------------- *)
Dummy := TRUE;

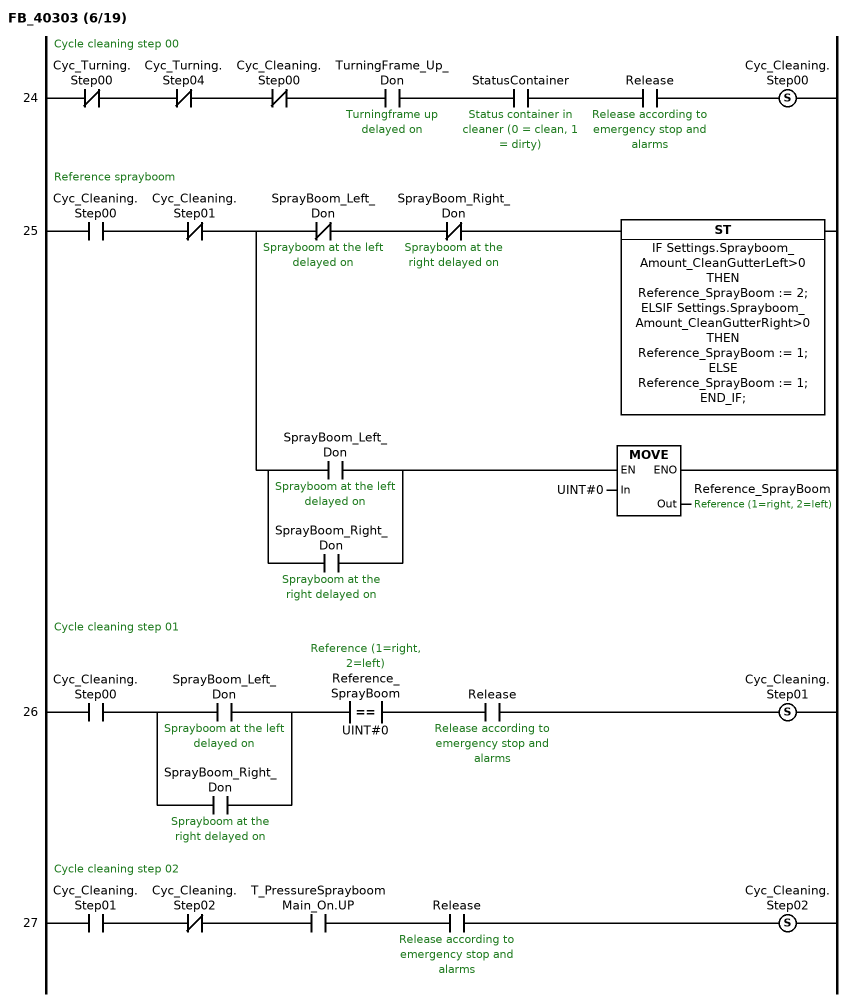
(* Rung 24: Cycle cleaning step 00 *)
IF NOT Cyc_Turning.Step00 AND NOT Cyc_Turning.Step04 AND NOT Cyc_Cleaning.Step00 AND TurningFrame_Up_Don AND StatusContainer AND Release THEN
    Cyc_Cleaning.Step00 := TRUE;
END_IF;
(* Rung 25: Reference sprayboom *)
IF Cyc_Cleaning.Step00 AND NOT Cyc_Cleaning.Step01 AND NOT SprayBoom_Left_Don AND NOT SprayBoom_Right_Don THEN
    IF Settings.Sprayboom_Amount_CleanGutterLeft>0 THEN
    	Reference_SprayBoom := 2;
    ELSIF Settings.Sprayboom_Amount_CleanGutterRight>0 THEN
    	Reference_SprayBoom := 1;
    ELSE
    	Reference_SprayBoom := 1;
    END_IF;
END_IF;
IF Cyc_Cleaning.Step00 AND NOT Cyc_Cleaning.Step01 AND (SprayBoom_Left_Don OR SprayBoom_Right_Don) THEN
    Reference_SprayBoom := UINT#0;
END_IF;
(* Rung 26: Cycle cleaning step 01 *)
IF Cyc_Cleaning.Step00 AND (SprayBoom_Left_Don OR SprayBoom_Right_Don) AND (Reference_SprayBoom = UINT#0) AND Release THEN
    Cyc_Cleaning.Step01 := TRUE;
END_IF;
(* Rung 27: Cycle cleaning step 02 *)
IF Cyc_Cleaning.Step01 AND NOT Cyc_Cleaning.Step02 AND T_PressureSprayboomMain_On.UP AND Release THEN
    Cyc_Cleaning.Step02 := TRUE;
END_IF;

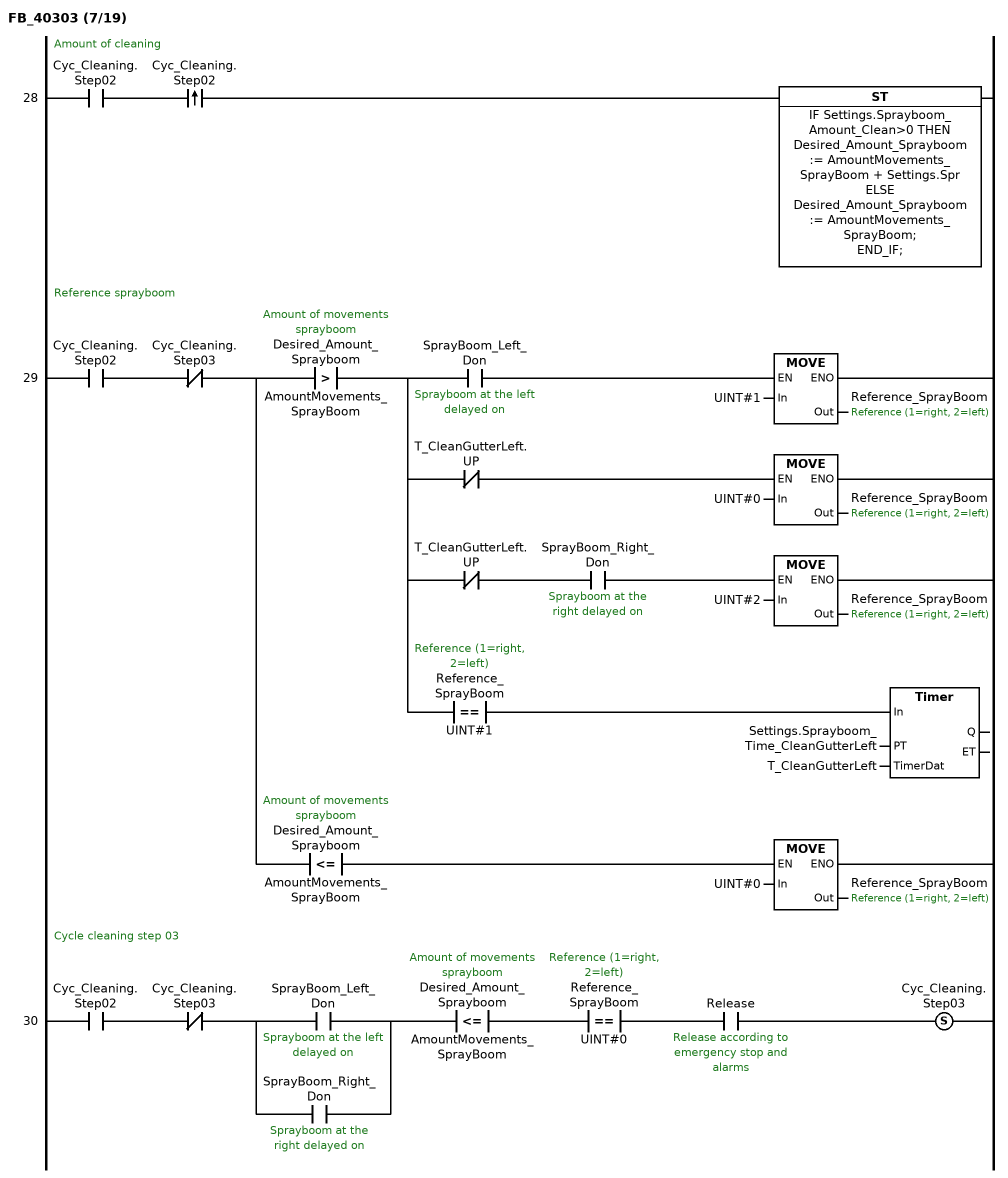
(* Rung 28: Amount of cleaning *)
_e6(CLK := Cyc_Cleaning.Step02);
IF Cyc_Cleaning.Step02 AND _e6.Q THEN
    IF Settings.Sprayboom_Amount_Clean>0 THEN
    	Desired_Amount_Sprayboom := AmountMovements_SprayBoom + Settings.Sprayboom_Amount_CleanGutterLeft;
    ELSE
    	Desired_Amount_Sprayboom := AmountMovements_SprayBoom;
    END_IF;
END_IF;
(* Rung 29: Reference sprayboom *)
_p7 := Cyc_Cleaning.Step02 AND NOT Cyc_Cleaning.Step03 AND (Desired_Amount_Sprayboom > AmountMovements_SprayBoom);
IF _p7 AND SprayBoom_Left_Don THEN Reference_SprayBoom := UINT#1; END_IF;
IF _p7 AND NOT T_CleanGutterLeft.UP THEN Reference_SprayBoom := UINT#0; END_IF;
IF _p7 AND NOT T_CleanGutterLeft.UP AND SprayBoom_Right_Don THEN Reference_SprayBoom := UINT#2; END_IF;
_t8 := Timer(In := _p7 AND (Reference_SprayBoom = UINT#1), PT := Settings.Sprayboom_Time_CleanGutterLeft, TimerDat := T_CleanGutterLeft);
IF Cyc_Cleaning.Step02 AND NOT Cyc_Cleaning.Step03 AND (Desired_Amount_Sprayboom <= AmountMovements_SprayBoom) THEN
    Reference_SprayBoom := UINT#0;
END_IF;
(* Rung 30: Cycle cleaning step 03 *)
IF Cyc_Cleaning.Step02 AND NOT Cyc_Cleaning.Step03 AND (SprayBoom_Left_Don OR SprayBoom_Right_Don) AND (Desired_Amount_Sprayboom <= AmountMovements_SprayBoom) AND (Reference_SprayBoom = UINT#0) AND Release THEN
    Cyc_Cleaning.Step03 := TRUE;
END_IF;

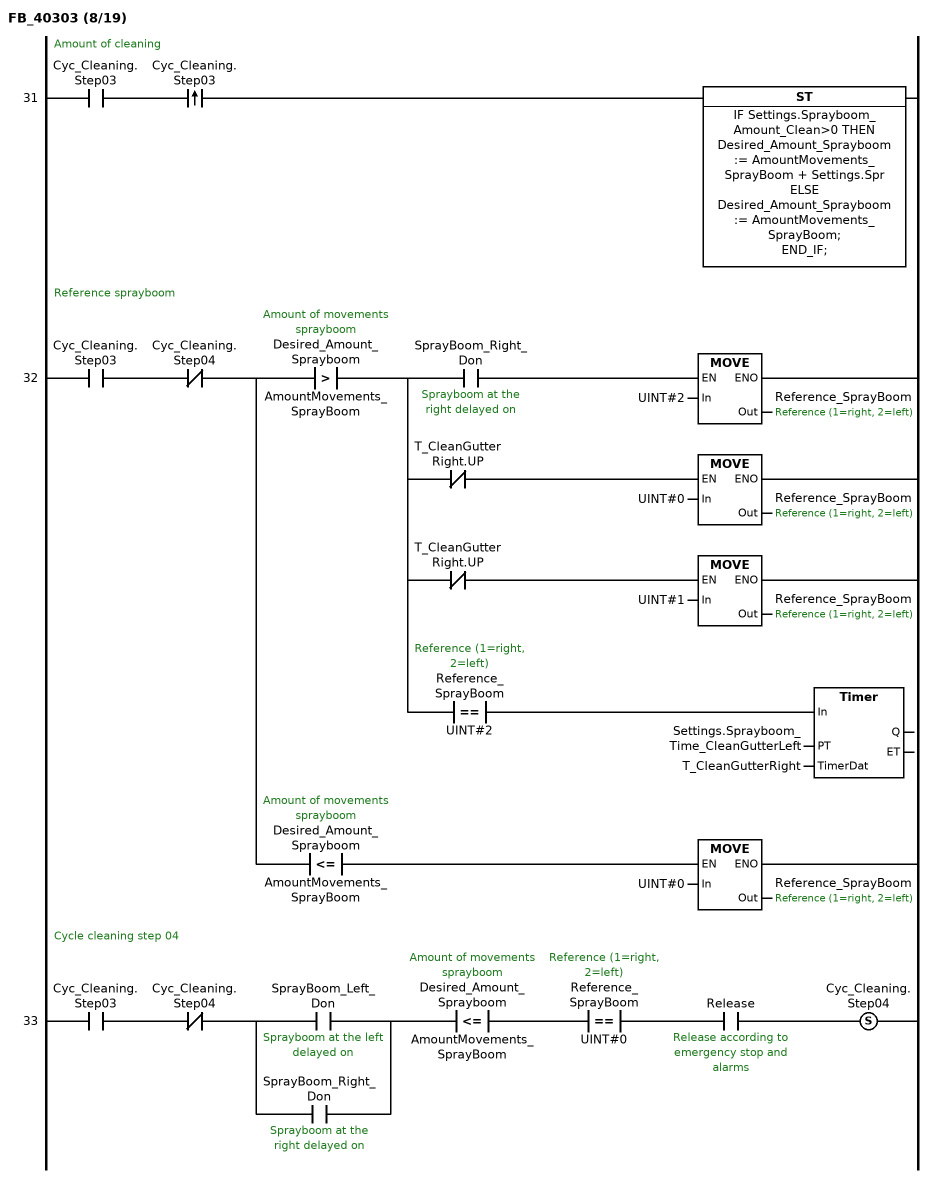
(* Rung 31: Amount of cleaning *)
_e9(CLK := Cyc_Cleaning.Step03);
IF Cyc_Cleaning.Step03 AND _e9.Q THEN
    IF Settings.Sprayboom_Amount_Clean>0 THEN
    	Desired_Amount_Sprayboom := AmountMovements_SprayBoom + Settings.Sprayboom_Amount_CleanGutterRight;
    ELSE
    	Desired_Amount_Sprayboom := AmountMovements_SprayBoom;
    END_IF;
END_IF;
(* Rung 32: Reference sprayboom *)
_p10 := Cyc_Cleaning.Step03 AND NOT Cyc_Cleaning.Step04 AND (Desired_Amount_Sprayboom > AmountMovements_SprayBoom);
IF _p10 AND SprayBoom_Right_Don THEN Reference_SprayBoom := UINT#2; END_IF;
IF _p10 AND NOT T_CleanGutterRight.UP THEN
    Reference_SprayBoom := UINT#0;
    Reference_SprayBoom := UINT#1;
END_IF;
_t11 := Timer(In := _p10 AND (Reference_SprayBoom = UINT#2), PT := Settings.Sprayboom_Time_CleanGutterLeft, TimerDat := T_CleanGutterRight);
IF Cyc_Cleaning.Step03 AND NOT Cyc_Cleaning.Step04 AND (Desired_Amount_Sprayboom <= AmountMovements_SprayBoom) THEN
    Reference_SprayBoom := UINT#0;
END_IF;
(* Rung 33: Cycle cleaning step 04 *)
IF Cyc_Cleaning.Step03 AND NOT Cyc_Cleaning.Step04 AND (SprayBoom_Left_Don OR SprayBoom_Right_Don) AND (Desired_Amount_Sprayboom <= AmountMovements_SprayBoom) AND (Reference_SprayBoom = UINT#0) AND Release THEN
    Cyc_Cleaning.Step04 := TRUE;
END_IF;

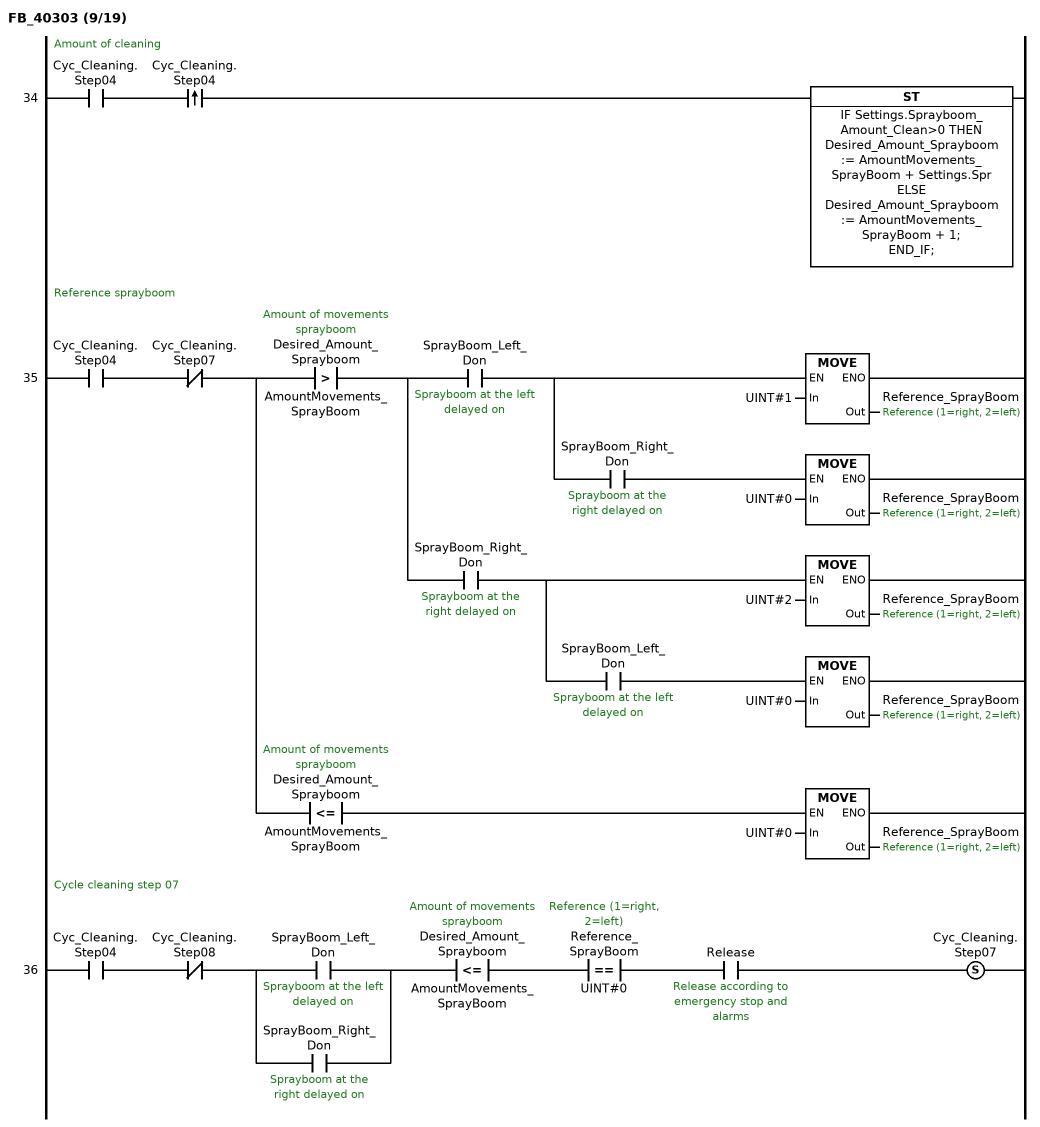
(* Rung 34: Amount of cleaning *)
_e12(CLK := Cyc_Cleaning.Step04);
IF Cyc_Cleaning.Step04 AND _e12.Q THEN
    IF Settings.Sprayboom_Amount_Clean>0 THEN
    	Desired_Amount_Sprayboom := AmountMovements_SprayBoom + Settings.Sprayboom_Amount_Clean;
    ELSE
    	Desired_Amount_Sprayboom := AmountMovements_SprayBoom + 1;
    END_IF;
END_IF;
(* Rung 35: Reference sprayboom *)
_p13 := Cyc_Cleaning.Step04 AND NOT Cyc_Cleaning.Step07 AND (Desired_Amount_Sprayboom > AmountMovements_SprayBoom);
IF _p13 AND SprayBoom_Left_Don THEN Reference_SprayBoom := UINT#1; END_IF;
IF _p13 AND SprayBoom_Left_Don AND SprayBoom_Right_Don THEN Reference_SprayBoom := UINT#0; END_IF;
IF _p13 AND SprayBoom_Right_Don THEN Reference_SprayBoom := UINT#2; END_IF;
IF _p13 AND SprayBoom_Right_Don AND SprayBoom_Left_Don THEN Reference_SprayBoom := UINT#0; END_IF;
IF Cyc_Cleaning.Step04 AND NOT Cyc_Cleaning.Step07 AND (Desired_Amount_Sprayboom <= AmountMovements_SprayBoom) THEN
    Reference_SprayBoom := UINT#0;
END_IF;
(* Rung 36: Cycle cleaning step 07 *)
IF Cyc_Cleaning.Step04 AND NOT Cyc_Cleaning.Step08 AND (SprayBoom_Left_Don OR SprayBoom_Right_Don) AND (Desired_Amount_Sprayboom <= AmountMovements_SprayBoom) AND (Reference_SprayBoom = UINT#0) AND Release THEN
    Cyc_Cleaning.Step07 := TRUE;
END_IF;

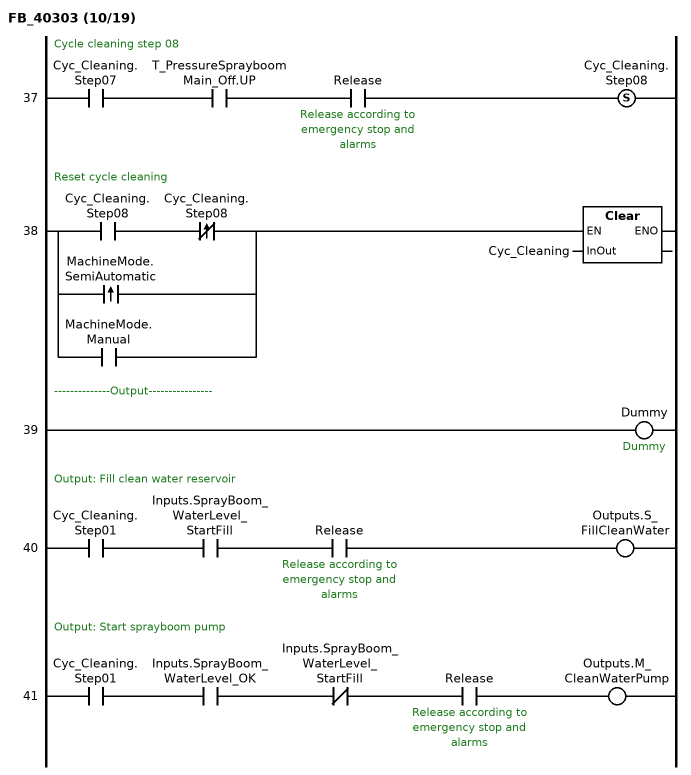
(* Rung 37: Cycle cleaning step 08 *)
IF Cyc_Cleaning.Step07 AND T_PressureSprayboomMain_Off.UP AND Release THEN
    Cyc_Cleaning.Step08 := TRUE;
END_IF;
(* Rung 38: Reset cycle cleaning *)
_e14(CLK := Cyc_Cleaning.Step08);
_e15(CLK := MachineMode.SemiAutomatic);
IF (Cyc_Cleaning.Step08 AND NOT _e14.Q) OR _e15.Q OR MachineMode.Manual THEN
    Clear(InOut := Cyc_Cleaning);
END_IF;
(* Rung 39: --------------Output---------------- *)
Dummy := TRUE;
(* Rung 40: Output: Fill clean water reservoir *)
Outputs.S_FillCleanWater := Cyc_Cleaning.Step01 AND Inputs.SprayBoom_WaterLevel_StartFill AND Release;
(* Rung 41: Output: Start sprayboom pump *)
Outputs.M_CleanWaterPump := Cyc_Cleaning.Step01 AND Inputs.SprayBoom_WaterLevel_OK AND NOT Inputs.SprayBoom_WaterLevel_StartFill AND Release;

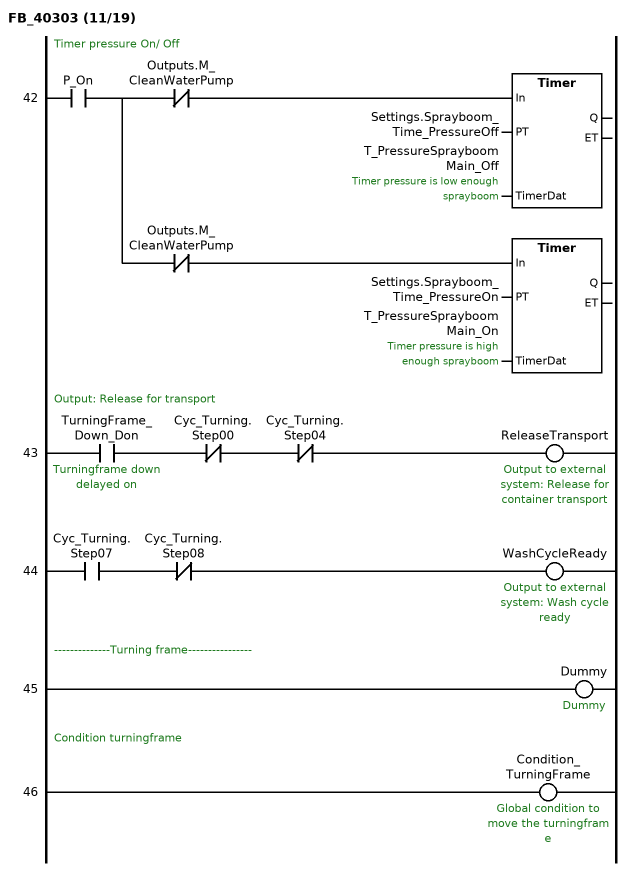
(* Rung 42: Timer pressure On/ Off *)
_t16 := Timer(In := P_On AND NOT Outputs.M_CleanWaterPump, PT := Settings.Sprayboom_Time_PressureOff, TimerDat := T_PressureSprayboomMain_Off);
_t17 := Timer(In := P_On AND NOT Outputs.M_CleanWaterPump, PT := Settings.Sprayboom_Time_PressureOn, TimerDat := T_PressureSprayboomMain_On);
(* Rung 43: Output: Release for transport *)
ReleaseTransport := TurningFrame_Down_Don AND NOT Cyc_Turning.Step00 AND NOT Cyc_Turning.Step04;
(* Rung 44 *)
WashCycleReady := Cyc_Turning.Step07 AND NOT Cyc_Turning.Step08;
(* Rung 45: --------------Turning frame---------------- *)
Dummy := TRUE;
(* Rung 46: Condition turningframe *)
Condition_TurningFrame := TRUE;

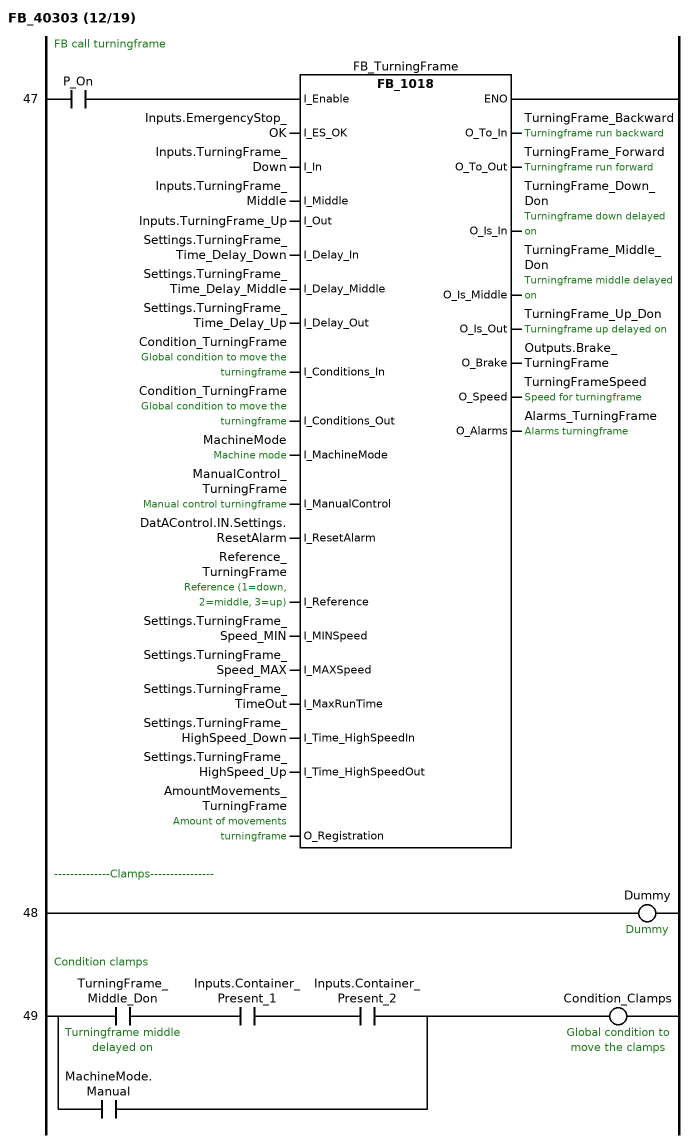
(* Rung 47: FB call turningframe *)
FB_TurningFrame(I_Enable := P_On, I_ES_OK := Inputs.EmergencyStop_OK, I_In := Inputs.TurningFrame_Down, I_Middle := Inputs.TurningFrame_Middle, I_Out := Inputs.TurningFrame_Up, I_Delay_In := Settings.TurningFrame_Time_Delay_Down, I_Delay_Middle := Settings.TurningFrame_Time_Delay_Middle, I_Delay_Out := Settings.TurningFrame_Time_Delay_Up, I_Conditions_In := Condition_TurningFrame, I_Conditions_Out := Condition_TurningFrame, I_MachineMode := MachineMode, I_ManualControl := ManualControl_TurningFrame, I_ResetAlarm := DatAControl.IN.Settings.ResetAlarm, I_Reference := Reference_TurningFrame, I_MINSpeed := Settings.TurningFrame_Speed_MIN, I_MAXSpeed := Settings.TurningFrame_Speed_MAX, I_MaxRunTime := Settings.TurningFrame_TimeOut, I_Time_HighSpeedIn := Settings.TurningFrame_HighSpeed_Down, I_Time_HighSpeedOut := Settings.TurningFrame_HighSpeed_Up, O_Registration := AmountMovements_TurningFrame, O_To_In => TurningFrame_Backward, O_To_Out => TurningFrame_Forward, O_Is_In => TurningFrame_Down_Don, O_Is_Middle => TurningFrame_Middle_Don, O_Is_Out => TurningFrame_Up_Don, O_Brake => Outputs.Brake_TurningFrame, O_Speed => TurningFrameSpeed, O_Alarms => Alarms_TurningFrame);
(* Rung 48: --------------Clamps---------------- *)
Dummy := TRUE;
(* Rung 49: Condition clamps *)
Condition_Clamps := (TurningFrame_Middle_Don AND Inputs.Container_Present_1 AND Inputs.Container_Present_2) OR MachineMode.Manual;

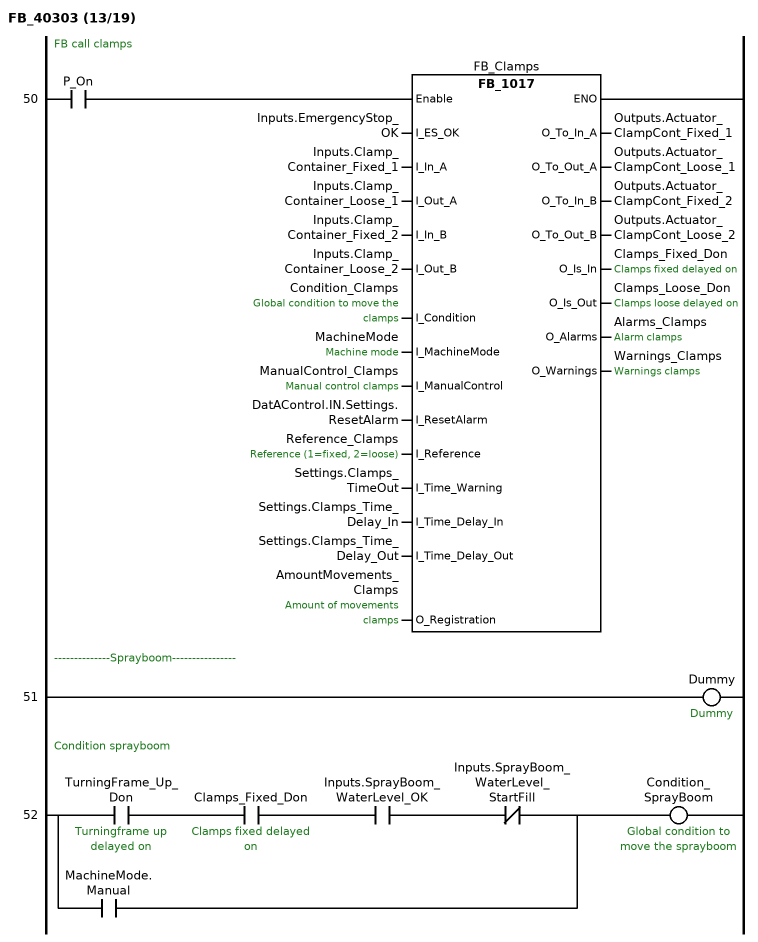
(* Rung 50: FB call clamps *)
FB_Clamps(Enable := P_On, I_ES_OK := Inputs.EmergencyStop_OK, I_In_A := Inputs.Clamp_Container_Fixed_1, I_Out_A := Inputs.Clamp_Container_Loose_1, I_In_B := Inputs.Clamp_Container_Fixed_2, I_Out_B := Inputs.Clamp_Container_Loose_2, I_Condition := Condition_Clamps, I_MachineMode := MachineMode, I_ManualControl := ManualControl_Clamps, I_ResetAlarm := DatAControl.IN.Settings.ResetAlarm, I_Reference := Reference_Clamps, I_Time_Warning := Settings.Clamps_TimeOut, I_Time_Delay_In := Settings.Clamps_Time_Delay_In, I_Time_Delay_Out := Settings.Clamps_Time_Delay_Out, O_Registration := AmountMovements_Clamps, O_To_In_A => Outputs.Actuator_ClampCont_Fixed_1, O_To_Out_A => Outputs.Actuator_ClampCont_Loose_1, O_To_In_B => Outputs.Actuator_ClampCont_Fixed_2, O_To_Out_B => Outputs.Actuator_ClampCont_Loose_2, O_Is_In => Clamps_Fixed_Don, O_Is_Out => Clamps_Loose_Don, O_Alarms => Alarms_Clamps, O_Warnings => Warnings_Clamps);
(* Rung 51: --------------Sprayboom---------------- *)
Dummy := TRUE;
(* Rung 52: Condition sprayboom *)
Condition_SprayBoom := (TurningFrame_Up_Don AND Clamps_Fixed_Don AND Inputs.SprayBoom_WaterLevel_OK AND NOT Inputs.SprayBoom_WaterLevel_StartFill) OR MachineMode.Manual;

